FUNCTION_BLOCK "FB_SafetyGroup"   // FB5, SCL
{ S7_Optimized_Access := 'TRUE' }
VERSION : 0.1
   VAR_INPUT
      bSafetySw : Bool;   // Normal close safety switch
      bRelayState : Bool;   // Safety relay feedback state
      bReset : Bool;   // Restore safety if raise this input
   END_VAR
   VAR_OUTPUT
      bMutingCtrl : Bool;   // Switch on before reset
      bResetCtrl : Bool;
      bSafetySw_Al : Bool;
      bReadyToReset : Bool;
      bResetAlarm : Bool;   // Set on when relay not turns on after reset
      bSafetyRelayAlarm : Bool;   // Set on when relay stays on when safety switch is activated
      bSafetyOK : Bool;
   END_VAR
   VAR
      fbResetPulse : TP_TIME;
      fbMutingPulse : TP_TIME;
   END_VAR
   VAR CONSTANT
      tResetTime : Time := T#1000ms;   // Reset time
      tMutingTime : Time := T#500ms;   // Muting time
   END_VAR
BEGIN
   IF #bReset THEN
       #bReadyToReset := FALSE;
       #bSafetySw_Al := FALSE;
       #bSafetyRelayAlarm := FALSE;
   END_IF;

   IF NOT #bSafetySw THEN
       #bSafetySw_Al := TRUE;
   END_IF;

   IF NOT #bSafetySw AND #bRelayState THEN
       #bSafetyRelayAlarm := TRUE;
   END_IF;

   IF #bSafetySw AND NOT #bRelayState THEN
       #bReadyToReset:=TRUE;
   END_IF;

   IF #bResetCtrl AND NOT #bMutingCtrl AND NOT #bRelayState THEN
       #bSafetyRelayAlarm := TRUE;
   END_IF;

   #fbResetPulse(IN:=#bSafetySw AND #bReset,
                 PT:=#tResetTime,
                 Q=>#bResetCtrl);

   #fbMutingPulse(IN:=#bSafetySw AND #bReset,
                  PT:=#tMutingTime,
                  Q=>#bMutingCtrl);

   #bSafetyOK := NOT #bSafetySw_Al AND #bSafetySw AND #bRelayState AND NOT #bResetCtrl AND NOT #bMutingCtrl;
END_FUNCTION_BLOCK

ORGANIZATION_BLOCK "FS_Safety"   // OB124, SCL, ProgramCycle
TITLE = "Main Program Sweep (Cycle)"
{ S7_Optimized_Access := 'TRUE' }
VERSION : 0.1
   VAR_INPUT
      Initial_Call : Bool;   // Initial call of this OB
      Remanence : Bool;   // =True, if remanent data are available
   END_VAR
   VAR_TEMP
      bStartPwr : Bool;
   END_VAR
BEGIN
   //Fail-safety control function block
   "FB_SafetyGroup_DB"(
                       //Switch state
                       bSafetySw:="bFS_MDB_SB1_St" AND "bFS_SR1_St" AND"bFS_SR1_1_St"AND
                       "bFS_SR1_2_St"AND"bFS_SR1_3_St"AND"bFS_SR2_St"AND
                       "bFS_SR2_1_St"AND"bFS_SR2_2_St"AND"bFS_SR2_3_St"AND
                       "bFS_SDB_SB2_St" AND"bFS_SR3_St"AND
                       "bFS_SR3_1_St"AND"bFS_SR3_2_St"AND"bFS_SR3_3_St"AND
                       "bFS_SB4_St"AND"bFS_SB5_St"AND"bFS_SB6_St"AND
                       "bFS_SB7_St"AND"bFS_PU_SB3_St",
                       //FS-relays feedback state
                       bRelayState:="bFS_MDB_KSF1_St" AND "bFS_MDB_KSF2_St" AND
                       "bFS_MDB_KSF3_St" AND "bFS_SDB_KSF1_St",
                       //Reset buttons
                       bReset:="bFS_MDB_SBR1_St" OR "bFS_SDB_SBR1_St" OR "bFS_PU_SBR1_St");

   //Fail-safety system alarm indication
   "bFS_MDB_SafetyAlarm_Ind" :=
   "bFS_SDB_SafetyAlarm_Ind" :=
   "bFS_PU_SafetyAlarm_Ind" := "FB_SafetyGroup_DB".bSafetySw_Al OR "FB_SafetyGroup_DB".bResetAlarm OR "FB_SafetyGroup_DB".bSafetyRelayAlarm;

   //Ready to reset. Reset buttons backlight
   "bFS_MDB_SBR1_HL" :=
   "bFS_SDB_SBR1_HL" :=
   "bFS_PU_SBR1_HL" := "FB_SafetyGroup_DB".bReadyToReset;

   //Muting control
   "bFS_MDB_SafetyMuting" := 
   "bFS_SDB_SafetyMuting" := "FB_SafetyGroup_DB".bMutingCtrl;

   //Reset fail safety
   "bFS_MDB_KSF1_2_Reset" :=
   "bFS_MDB_KSF3_Reset" :=
   "bFS_Lift2Safety_Reset" :=
   "bFS_StackerSafety_Reset" :=
   "bFS_SDB_KSF1_Reset":=
   "bFS_Lift1Safety_Reset":="FB_SafetyGroup_DB".bResetCtrl;

   //Soft start power
   "FB_StartTimer_DB".TON(IN:="FB_SafetyGroup_DB".bSafetyOK AND NOT #bStartPwr,
                          PT:=t#500ms);
   IF "FB_StartTimer_DB".Q THEN
       #bStartPwr := true;
   END_IF;

   "FB_Station1Pwr_DB"(bOn := "FB_SafetyGroup_DB".bSafetyOK,
                       bState := "bStation1_Pwr_St",
                       bReset := "bResetAlarm",
                       bCtrl => "bStation1_Pwr_Ctrl",
                       bStart := #bStartPwr);

   "FB_Station2Pwr_DB"(bOn := "FB_SafetyGroup_DB".bSafetyOK,
                       bState := "bStation2_Pwr_St",
                       bReset := "bResetAlarm",
                       bCtrl => "bStation2_Pwr_Ctrl",
                       bStart := #bStartPwr);

   "FB_Station3Pwr_DB"(bOn := "FB_SafetyGroup_DB".bSafetyOK,
                       bState := "bStation3_Pwr_St",
                       bReset := "bResetAlarm",
                       bCtrl => "bStation3_Pwr_Ctrl",
                       bStart := #bStartPwr);

   "FB_Station4Pwr_DB"(bOn := "FB_SafetyGroup_DB".bSafetyOK,
                       bState := "bStation4_Pwr_St",
                       bReset := "bResetAlarm",
                       bCtrl => "bStation4_Pwr_Ctrl",
                       bStart := #bStartPwr);

   "FB_Station5Pwr_DB"(bOn := "FB_SafetyGroup_DB".bSafetyOK,
                       bState := "bStation5_Pwr_St",
                       bReset := "bResetAlarm",
                       bCtrl => "bStation5_Pwr_Ctrl",
                       bStart := #bStartPwr);

   "FB_Station6Pwr_DB"(bOn := "FB_SafetyGroup_DB".bSafetyOK,
                       bState := "bStation6_Pwr_St",
                       bReset := "bResetAlarm",
                       bCtrl => "bStation6_Pwr_Ctrl",
                       bStart := #bStartPwr);

   "FB_Station7Pwr_DB"(bOn := "FB_SafetyGroup_DB".bSafetyOK,
                       bState := "bStation7_Pwr_St",
                       bReset := "bResetAlarm",
                       bCtrl => "bStation7_Pwr_Ctrl",
                       bStart := #bStartPwr);

   "FB_Station8Pwr_DB"(bOn := "FB_SafetyGroup_DB".bSafetyOK,
                       bState := "bStation8_Pwr_St",
                       bReset := "bResetAlarm",
                       bCtrl => "bStation8_Pwr_Ctrl",
                       bStart := #bStartPwr);

   "FB_Station9Pwr_DB"(bOn := "FB_SafetyGroup_DB".bSafetyOK,
                       bState := "bStation9_Pwr_St",
                       bReset := "bResetAlarm",
                       bCtrl => "bStation9_Pwr_Ctrl",
                       bStart := #bStartPwr);

   "FB_Station10Pwr_DB"(bOn := "FB_SafetyGroup_DB".bSafetyOK,
                        bState := "bStation10_Pwr_St",
                        bReset := "bResetAlarm",
                        bCtrl => "bStation10_Pwr_Ctrl",
                        bStart := #bStartPwr);

   "FB_Station11Pwr_DB"(bOn := "FB_SafetyGroup_DB".bSafetyOK,
                        bState := "bStation11_Pwr_St",
                        bReset := "bResetAlarm",
                        bCtrl => "bStation11_Pwr_Ctrl",
                        bStart := #bStartPwr);

   "FB_Station12Pwr_DB"(bOn := "FB_SafetyGroup_DB".bSafetyOK,
                        bState := "bStation12_Pwr_St",
                        bReset := "bResetAlarm",
                        bCtrl => "bStation12_Pwr_Ctrl",
                        bStart := #bStartPwr);

   "FB_Station13Pwr_DB"(bOn := "FB_SafetyGroup_DB".bSafetyOK,
                        bState := "bStation13_Pwr_St",
                        bReset := "bResetAlarm",
                        bCtrl => "bStation13_Pwr_Ctrl",
                        bStart := #bStartPwr);

   "FB_Station14Pwr_DB"(bOn := "FB_SafetyGroup_DB".bSafetyOK,
                        bState := "bStation14_Pwr_St",
                        bReset := "bResetAlarm",
                        bCtrl => "bStation14_Pwr_Ctrl",
                        bStart := #bStartPwr);

   "FB_Conv35_36Pwr_DB"(bOn := "FB_SafetyGroup_DB".bSafetyOK,
                        bState := "bConv35_36_Pwr_St",
                        bReset := "bResetAlarm",
                        bCtrl => "bConv35_36_Pwr_Ctrl",
                        bStart := #bStartPwr);

   "FB_SDB_KM1Pwr_DB"(bOn := "FB_SafetyGroup_DB".bSafetyOK,
                      bState := "bSDB_KM1_St",
                        bReset := "bResetAlarm",
                        bCtrl => "bSDB_KM1_Ctrl",
                        bStart := #bStartPwr);
END_ORGANIZATION_BLOCK

// folder: Safety/PWR

FUNCTION_BLOCK "FB_PowerGroup"   // FB4, SCL
{ S7_Optimized_Access := 'TRUE' }
VERSION : 0.1
   VAR_INPUT
      bOn : Bool;
      bState : Bool;
      bReset : Bool;
   END_VAR
   VAR_OUTPUT
      bCtrl : Bool;
      bAlarm : Bool;
      bRelayOnAlarm : Bool;
      bRelayOffAlarm : Bool;
   END_VAR
   VAR_IN_OUT
      bStart : Bool;
   END_VAR
   VAR
      fbRestartDelay : TOF_TIME;
      fbOnAlarm : TON_TIME;
      fbOffAlarm : TON_TIME;
   END_VAR
   VAR CONSTANT
      tAlarmDelay : Time := T#5000ms;   // Alarm Delay
      tRestartDelay : Time := T#1000ms;   // Restart Delay
   END_VAR
BEGIN


   IF #bReset THEN
       #bRelayOnAlarm := false;
       #bRelayOffAlarm := false;
   END_IF;

   #fbRestartDelay(IN:=#bCtrl,
                   PT:=#tRestartDelay);

   #fbOffAlarm(IN:=NOT #bCtrl AND #bState,
               PT:=#tAlarmDelay);
   IF #fbOffAlarm.Q THEN
       #bRelayOffAlarm := true;
   END_IF;


   #fbOnAlarm(IN := #bCtrl AND NOT #bState,
               PT := #tAlarmDelay);
    IF #fbOnAlarm.Q THEN
        #bRelayOnAlarm := true;
    END_IF;


   #bAlarm := #bRelayOffAlarm OR #bRelayOnAlarm;

   IF #bAlarm THEN
       #bCtrl := false;
   ELSE
       IF #bOn THEN
           IF NOT #fbRestartDelay.Q THEN
               IF #bStart AND NOT #bCtrl THEN
                   #bCtrl := true;
                   #bStart := false;
               END_IF;
           END_IF;
       ELSE
           #bCtrl := false;
       END_IF;
   END_IF;
END_FUNCTION_BLOCK